//读取叠台的数据
rtRead(CLK:=ReadPointVelues , Q=> );
ftRead(CLK:=ReadPointVelues , Q=> );	
	IF rtRead.Q THEN
		mcReadMotionFunctionValues.Execute:=TRUE;
		CamTable3.pArray:=ADR(arrTableData);
		CamTable3.ArraySize:=SIZEOF(arrTableData);
		CamTable3.NoOfColumns:=2;
		CamTable3.NoOfRows:=3601;
		CamTable3.TableType:=10;	
	END_IF	
	 mcReadMotionFunctionValues1(
		  Execute:=                          mcReadMotionFunctionValues.Execute , 
		  CamTableID:=                   iTable , 
		  ValueSelectMask:=               1 ,
		  StartPosMaster:=               0 , 
		  EndPosMaster:=                360 , //360
		  Increment:=                       0.1 , 
		  Done=>                           arrReadPosDone , 
		  Busy=>mcReadMotionFunctionValues_Busy                              , 
		  Error=>mcReadMotionFunctionValues_Error                             , 
		  ErrorID=>mcReadMotionFunctionValues_ErrorID                         , 
		  CamTable:=                      CamTable3      );
	IF ftRead.Q THEN
		mcReadMotionFunctionValues.Execute:=FALSE;	
	END_IF	
//叠台中心点，主轴相位计算 fbCenterPoint
	Test_int:=REAL_TO_INT(fMainPos*10);
	FOR	i:=0 TO Test_int BY 1  DO
		IF (fbCenterPoint-0.15)< arrTableData[i,1] AND arrTableData[i,1]<(fbCenterPoint +0.15) THEN
			iFend:=i;
			Master_MidPos:=arrTableData[i,0];			
		END_IF		
	END_FOR
END_ACTION

ACTION Motion:
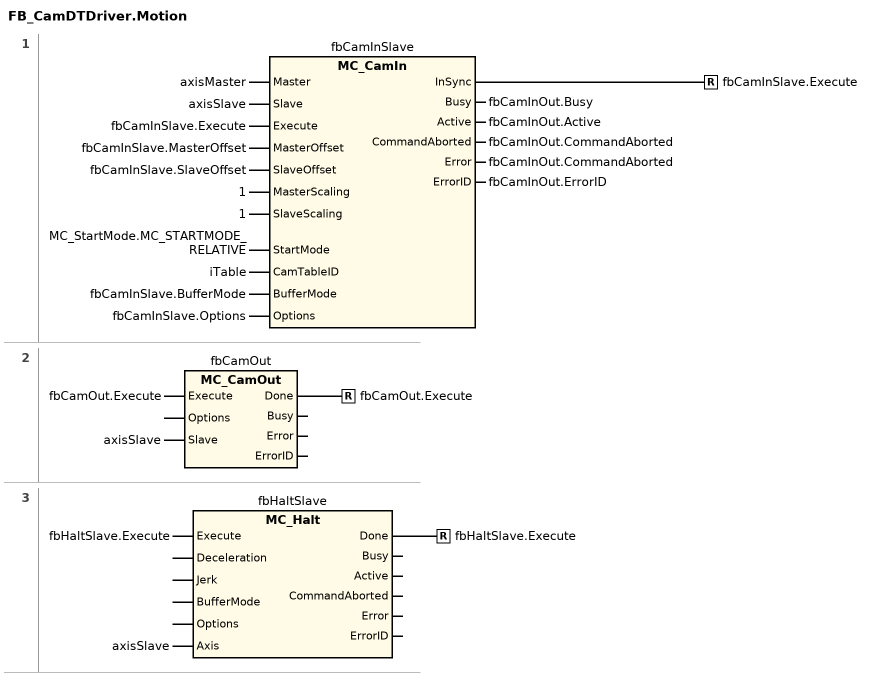
// NETWORK 1
fbCamInSlave(
    Master := axisMaster,
    Slave := axisSlave,
    Execute := fbCamInSlave.Execute,
    MasterOffset := fbCamInSlave.MasterOffset,
    SlaveOffset := fbCamInSlave.SlaveOffset,
    MasterScaling := 1,
    SlaveScaling := 1,
    StartMode := MC_StartMode.MC_STARTMODE_RELATIVE,
    CamTableID := iTable,
    BufferMode := fbCamInSlave.BufferMode,
    Options := fbCamInSlave.Options,
    Busy => fbCamInOut.Busy,
    Active => fbCamInOut.Active,
    CommandAborted => fbCamInOut.CommandAborted,
    Error => fbCamInOut.CommandAborted,
    ErrorID => fbCamInOut.ErrorID); // MC_CamIn
fbCamInSlave.Execute R= fbCamInSlave.InSync;

// NETWORK 2
fbCamOut(Execute := fbCamOut.Execute, Slave := axisSlave); // MC_CamOut
fbCamOut.Execute R= fbCamOut.Done;

// NETWORK 3
fbHaltSlave(Execute := fbHaltSlave.Execute, Axis := axisSlave); // MC_Halt
fbHaltSlave.Execute R= fbHaltSlave.Done;
END_ACTION

END_FUNCTION_BLOCK

// ---- P2POUs/BasicFunction/12_User2/FB_Rectify.TcPOU
FUNCTION_BLOCK FB_Rectify
VAR_INPUT
	
END_VAR
VAR_IN_OUT
     RecCtrl:     ST_RecCtrl;
END_VAR
VAR
   rtRec  :ARRAY[1..4] OF Tc2_Standard.R_TRIG;
END_VAR









rtRec[1](CLK:=RecCtrl.Cmd.bLock , Q=> );
rtRec[2](CLK:=RecCtrl.Cmd.bAuto , Q=> );
rtRec[3](CLK:=RecCtrl.Cmd.bManual , Q=> );
rtRec[4](CLK:=RecCtrl.Cmd.bCentre , Q=> );

IF rtRec[1].Q   THEN  //外部锁定
    RecCtrl.Io.boLock:=TRUE;
    RecCtrl.Io.boAuto:=FALSE;
    RecCtrl.Io.boManual:=FALSE;
    RecCtrl.Io.boCentre:=FALSE;
END_IF

IF rtRec[2].Q   THEN  //自动
    RecCtrl.Io.boLock:=FALSE;
    RecCtrl.Io.boAuto:=TRUE;
    RecCtrl.Io.boManual:=FALSE;
    RecCtrl.Io.boCentre:=FALSE;
END_IF

IF rtRec[3].Q   THEN  //手动
    RecCtrl.Io.boLock:=FALSE;
    RecCtrl.Io.boAuto:=FALSE;
    RecCtrl.Io.boManual:=TRUE;
    RecCtrl.Io.boCentre:=FALSE;
END_IF

IF rtRec[4].Q   THEN  //居中
    RecCtrl.Io.boLock:=FALSE;
    RecCtrl.Io.boAuto:=FALSE;
    RecCtrl.Io.boManual:=FALSE;
    RecCtrl.Io.boCentre:=TRUE;
END_IF


RecCtrl.Status.bError:=RecCtrl.Io.biError;
RecCtrl.Status.bRuning:=RecCtrl.Io.biCentre;

END_FUNCTION_BLOCK

// ---- P2POUs/BasicFunction/12_User2/Program_1.TcPOU
PROGRAM Program_1
VAR
Step0:INT;
TON1:Tc2_Standard.TON;
DemarcateStart,DemarcateDone,Demarcateing,CCDStart:BOOL;
	i: UINT;	
END_VAR

// scRecipe(iRecipe2:=iRecipe );
 
 TON1(IN:= , PT:=T#5S , Q=> , ET=> );//拍照延时复位


CASE Step0 OF
		0://等待CCD标定启动信号
		        P2M1_CCD.AnRec.Start.iPhotoDo:=0;
		        P2M1_CCD.AnRec.iDemarcatResult:=0;
			IF DemarcateStart THEN
				i:=0;//标定点位记数
			    P2M1_CCD.AnRec.Start.iPhotoDo:=1;
				DemarcateStart:=FALSE;//复位标定启动
				DemarcateDone:=FALSE;//CCD标定完成
				Demarcateing:=TRUE;//CCD标定中
				Step0:=5;
			END_IF
	5:
IF 		P2M1_CCD.AnRec.iDemarcatResult=1 AND  P2M1_CCD.AnRec.Start.iPhotoDo=0 THEN 
         P2M1_CCD.AnRec.iDemarcatResult:=0;
		 	i:=1;
			Step0:=10;
ELSIF 	P2M1_CCD.AnRec.iDemarcatResult=2 AND  P2M1_CCD.AnRec.Start.iPhotoDo=0 THEN 
	P2M1_CCD.AnRec.iDemarcatResult:=0;
	Step0:=999;
END_IF
		10://判断CCD标定走到第几个点位
					IF  i=1 THEN
									arrAxisPar[P2M1_Axise.AxisName.AndeviationX1].arrTargetPoint[3]:=arrAxisPar[P2M1_Axise.AxisName.AndeviationX1].arrTargetPoint[1];//+(103.94*COS(DEG_TO_RAD(CCD_W+225))-103.94*COS(DEG_TO_RAD(225))); 
									arrAxisPar[P2M1_Axise.AxisName.AndeviationX2].arrTargetPoint[3]:=arrAxisPar[P2M1_Axise.AxisName.AndeviationX2].arrTargetPoint[1];//+(103.94*SIN(DEG_TO_RAD(CCD_W+315))-103.94*COS(DEG_TO_RAD(315)));
									arrAxisPar[P2M1_Axise.AxisName.AndeviationY].arrTargetPoint[3]:=arrAxisPar[P2M1_Axise.AxisName.AndeviationY].arrTargetPoint[1];//+(103.94*COS(DEG_TO_RAD(CCD_W+135))-103.94*COS(DEG_TO_RAD(135)));	
									//i:=i+1;
									Step0:=20;
					ELSIF i=2 THEN
									arrAxisPar[P2M1_Axise.AxisName.AndeviationX1].arrTargetPoint[3]:=arrAxisPar[P2M1_Axise.AxisName.AndeviationX1].arrTargetPoint[1]+4;//+(103.94*COS(DEG_TO_RAD(CCD_W+225))-103.94*COS(DEG_TO_RAD(225))); 
									arrAxisPar[P2M1_Axise.AxisName.AndeviationX2].arrTargetPoint[3]:=arrAxisPar[P2M1_Axise.AxisName.AndeviationX2].arrTargetPoint[1]+4;//+(103.94*SIN(DEG_TO_RAD(CCD_W+315))-103.94*COS(DEG_TO_RAD(315)));
									arrAxisPar[P2M1_Axise.AxisName.AndeviationY].arrTargetPoint[3]:=arrAxisPar[P2M1_Axise.AxisName.AndeviationY].arrTargetPoint[1];//+(103.94*COS(DEG_TO_RAD(CCD_W+135))-103.94*COS(DEG_TO_RAD(135)));
									//i:=i+1;
									Step0:=20;
					ELSIF i=3 THEN
									arrAxisPar[P2M1_Axise.AxisName.AndeviationX1].arrTargetPoint[3]:=arrAxisPar[P2M1_Axise.AxisName.AndeviationX1].arrTargetPoint[1]+4;//+(103.94*COS(DEG_TO_RAD(CCD_W+225))-103.94*COS(DEG_TO_RAD(225))); 
									arrAxisPar[P2M1_Axise.AxisName.AndeviationX2].arrTargetPoint[3]:=arrAxisPar[P2M1_Axise.AxisName.AndeviationX2].arrTargetPoint[1]+4;//+(103.94*SIN(DEG_TO_RAD(CCD_W+315))-103.94*COS(DEG_TO_RAD(315)));
									arrAxisPar[P2M1_Axise.AxisName.AndeviationY].arrTargetPoint[3]:=arrAxisPar[P2M1_Axise.AxisName.AndeviationY].arrTargetPoint[1]+4;//+(103.94*COS(DEG_TO_RAD(CCD_W+135))-103.94*COS(DEG_TO_RAD(135)));	
									//i:=i+1;
									Step0:=20;									
					ELSIF i=4 THEN
								arrAxisPar[P2M1_Axise.AxisName.AndeviationX1].arrTargetPoint[3]:=arrAxisPar[P2M1_Axise.AxisName.AndeviationX1].arrTargetPoint[1];//+(103.94*COS(DEG_TO_RAD(CCD_W+225))-103.94*COS(DEG_TO_RAD(225))); 
								arrAxisPar[P2M1_Axise.AxisName.AndeviationX2].arrTargetPoint[3]:=arrAxisPar[P2M1_Axise.AxisName.AndeviationX2].arrTargetPoint[1];//+(103.94*SIN(DEG_TO_RAD(CCD_W+315))-103.94*COS(DEG_TO_RAD(315)));
								arrAxisPar[P2M1_Axise.AxisName.AndeviationY].arrTargetPoint[3]:=arrAxisPar[P2M1_Axise.AxisName.AndeviationY].arrTargetPoint[1]+4;//+(103.94*COS(DEG_TO_RAD(CCD_W+135))-103.94*COS(DEG_TO_RAD(135)));	
								//i:=i+1;
								Step0:=20;		
					ELSIF i=5 THEN
								arrAxisPar[P2M1_Axise.AxisName.AndeviationX1].arrTargetPoint[3]:=arrAxisPar[P2M1_Axise.AxisName.AndeviationX1].arrTargetPoint[1]-4;//+(103.94*COS(DEG_TO_RAD(CCD_W+225))-103.94*COS(DEG_TO_RAD(225))); 
								arrAxisPar[P2M1_Axise.AxisName.AndeviationX2].arrTargetPoint[3]:=arrAxisPar[P2M1_Axise.AxisName.AndeviationX2].arrTargetPoint[1]-4;//+(103.94*SIN(DEG_TO_RAD(CCD_W+315))-103.94*COS(DEG_TO_RAD(315)));
								arrAxisPar[P2M1_Axise.AxisName.AndeviationY].arrTargetPoint[3]:=arrAxisPar[P2M1_Axise.AxisName.AndeviationY].arrTargetPoint[1]+4;//+(103.94*COS(DEG_TO_RAD(CCD_W+135))-103.94*COS(DEG_TO_RAD(135)));	
							//	i:=i+1;
								Step0:=20;		
					ELSIF i=6 THEN
								arrAxisPar[P2M1_Axise.AxisName.AndeviationX1].arrTargetPoint[3]:=arrAxisPar[P2M1_Axise.AxisName.AndeviationX1].arrTargetPoint[1]-4;//+(103.94*COS(DEG_TO_RAD(CCD_W+225))-103.94*COS(DEG_TO_RAD(225))); 
								arrAxisPar[P2M1_Axise.AxisName.AndeviationX2].arrTargetPoint[3]:=arrAxisPar[P2M1_Axise.AxisName.AndeviationX2].arrTargetPoint[1]-4;//+(103.94*SIN(DEG_TO_RAD(CCD_W+315))-103.94*COS(DEG_TO_RAD(315)));
								arrAxisPar[P2M1_Axise.AxisName.AndeviationY].arrTargetPoint[3]:=arrAxisPar[P2M1_Axise.AxisName.AndeviationY].arrTargetPoint[1];//+(103.94*COS(DEG_TO_RAD(CCD_W+135))-103.94*COS(DEG_TO_RAD(135)));	
								//i:=i+1;
								Step0:=20;		
					ELSIF i=7 THEN
									arrAxisPar[P2M1_Axise.AxisName.AndeviationX1].arrTargetPoint[3]:=arrAxisPar[P2M1_Axise.AxisName.AndeviationX1].arrTargetPoint[1]-4;//+(103.94*COS(DEG_TO_RAD(CCD_W+225))-103.94*COS(DEG_TO_RAD(225))); 
									arrAxisPar[P2M1_Axise.AxisName.AndeviationX2].arrTargetPoint[3]:=arrAxisPar[P2M1_Axise.AxisName.AndeviationX2].arrTargetPoint[1]-4;//+(103.94*SIN(DEG_TO_RAD(CCD_W+315))-103.94*COS(DEG_TO_RAD(315)));
									arrAxisPar[P2M1_Axise.AxisName.AndeviationY].arrTargetPoint[3]:=arrAxisPar[P2M1_Axise.AxisName.AndeviationY].arrTargetPoint[1]-4;//+(103.94*COS(DEG_TO_RAD(CCD_W+135))-103.94*COS(DEG_TO_RAD(135)));
								//	i:=i+1;
									Step0:=20;		
					ELSIF i=8 THEN
									arrAxisPar[P2M1_Axise.AxisName.AndeviationX1].arrTargetPoint[3]:=arrAxisPar[P2M1_Axise.AxisName.AndeviationX1].arrTargetPoint[1];//+(103.94*COS(DEG_TO_RAD(CCD_W+225))-103.94*COS(DEG_TO_RAD(225))); 
									arrAxisPar[P2M1_Axise.AxisName.AndeviationX2].arrTargetPoint[3]:=arrAxisPar[P2M1_Axise.AxisName.AndeviationX2].arrTargetPoint[1];//+(103.94*SIN(DEG_TO_RAD(CCD_W+315))-103.94*COS(DEG_TO_RAD(315)));
									arrAxisPar[P2M1_Axise.AxisName.AndeviationY].arrTargetPoint[3]:=arrAxisPar[P2M1_Axise.AxisName.AndeviationY].arrTargetPoint[1]-4;//+(103.94*COS(DEG_TO_RAD(CCD_W+135))-103.94*COS(DEG_TO_RAD(135)));	
									//i:=i+1;
									Step0:=20;		
					ELSIF i=9 THEN
								arrAxisPar[P2M1_Axise.AxisName.AndeviationX1].arrTargetPoint[3]:=arrAxisPar[P2M1_Axise.AxisName.AndeviationX1].arrTargetPoint[1]+4;//+(103.94*COS(DEG_TO_RAD(CCD_W+225))-103.94*COS(DEG_TO_RAD(225))); 
								arrAxisPar[P2M1_Axise.AxisName.AndeviationX2].arrTargetPoint[3]:=arrAxisPar[P2M1_Axise.AxisName.AndeviationX2].arrTargetPoint[1]+4;//+(103.94*SIN(DEG_TO_RAD(CCD_W+315))-103.94*COS(DEG_TO_RAD(315)));
								arrAxisPar[P2M1_Axise.AxisName.AndeviationY].arrTargetPoint[3]:=arrAxisPar[P2M1_Axise.AxisName.AndeviationY].arrTargetPoint[1]-4;//+(103.94*COS(DEG_TO_RAD(CCD_W+135))-103.94*COS(DEG_TO_RAD(135)));	
								//i:=i+1;
								Step0:=20;		
					ELSIF i=10 THEN
								arrAxisPar[P2M1_Axise.AxisName.AndeviationX1].arrTargetPoint[3]:=arrAxisPar[P2M1_Axise.AxisName.AndeviationX1].arrTargetPoint[1];//+(103.94*COS(DEG_TO_RAD(CCD_W+225))-103.94*COS(DEG_TO_RAD(225))); 
								arrAxisPar[P2M1_Axise.AxisName.AndeviationX2].arrTargetPoint[3]:=arrAxisPar[P2M1_Axise.AxisName.AndeviationX2].arrTargetPoint[1];//+(103.94*SIN(DEG_TO_RAD(CCD_W+315))-103.94*COS(DEG_TO_RAD(315)));
								arrAxisPar[P2M1_Axise.AxisName.AndeviationY].arrTargetPoint[3]:=arrAxisPar[P2M1_Axise.AxisName.AndeviationY].arrTargetPoint[1];//+(103.94*COS(DEG_TO_RAD(CCD_W+135))-103.94*COS(DEG_TO_RAD(135)));	
								//i:=i+1;
								Step0:=20;		
					ELSIF i=11 THEN
								arrAxisPar[P2M1_Axise.AxisName.AndeviationX1].arrTargetPoint[3]:=arrAxisPar[P2M1_Axise.AxisName.AndeviationX1].arrTargetPoint[1]+(103.94*COS(DEG_TO_RAD(2+225))-103.94*COS(DEG_TO_RAD(225))); 
								arrAxisPar[P2M1_Axise.AxisName.AndeviationX2].arrTargetPoint[3]:=arrAxisPar[P2M1_Axise.AxisName.AndeviationX2].arrTargetPoint[1]+(103.94*SIN(DEG_TO_RAD(2+315))-103.94*COS(DEG_TO_RAD(315)));
								arrAxisPar[P2M1_Axise.AxisName.AndeviationY].arrTargetPoint[3]:=arrAxisPar[P2M1_Axise.AxisName.AndeviationY].arrTargetPoint[1]+(103.94*COS(DEG_TO_RAD(2+135))-103.94*COS(DEG_TO_RAD(135)));	
								//i:=i+1;
								Step0:=20;		
					ELSIF i=12 THEN
									arrAxisPar[P2M1_Axise.AxisName.AndeviationX1].arrTargetPoint[3]:=arrAxisPar[P2M1_Axise.AxisName.AndeviationX1].arrTargetPoint[1]+(103.94*COS(DEG_TO_RAD(1+225))-103.94*COS(DEG_TO_RAD(225))); 
									arrAxisPar[P2M1_Axise.AxisName.AndeviationX2].arrTargetPoint[3]:=arrAxisPar[P2M1_Axise.AxisName.AndeviationX2].arrTargetPoint[1]+(103.94*SIN(DEG_TO_RAD(1+315))-103.94*COS(DEG_TO_RAD(315)));
									arrAxisPar[P2M1_Axise.AxisName.AndeviationY].arrTargetPoint[3]:=arrAxisPar[P2M1_Axise.AxisName.AndeviationY].arrTargetPoint[1]+(103.94*COS(DEG_TO_RAD(1+135))-103.94*COS(DEG_TO_RAD(135)));
									//i:=i+1;
									Step0:=20;		
					
					ELSIF i=130 THEN
									arrAxisPar[P2M1_Axise.AxisName.AndeviationX1].arrTargetPoint[3]:=arrAxisPar[P2M1_Axise.AxisName.AndeviationX1].arrTargetPoint[1];//+(103.94*COS(DEG_TO_RAD(CCD_W+225))-103.94*COS(DEG_TO_RAD(225))); 
									arrAxisPar[P2M1_Axise.AxisName.AndeviationX2].arrTargetPoint[3]:=arrAxisPar[P2M1_Axise.AxisName.AndeviationX2].arrTargetPoint[1];//+(103.94*SIN(DEG_TO_RAD(CCD_W+315))-103.94*COS(DEG_TO_RAD(315)));
									arrAxisPar[P2M1_Axise.AxisName.AndeviationY].arrTargetPoint[3]:=arrAxisPar[P2M1_Axise.AxisName.AndeviationY].arrTargetPoint[1];//+(103.94*COS(DEG_TO_RAD(CCD_W+135))-103.94*COS(DEG_TO_RAD(135)));	
									//i:=i+1;
									Step0:=20;		
					ELSIF i=140 THEN
								arrAxisPar[P2M1_Axise.AxisName.AndeviationX1].arrTargetPoint[3]:=arrAxisPar[P2M1_Axise.AxisName.AndeviationX1].arrTargetPoint[1]+(103.94*COS(DEG_TO_RAD(-1+225))-103.94*COS(DEG_TO_RAD(225))); 
								arrAxisPar[P2M1_Axise.AxisName.AndeviationX2].arrTargetPoint[3]:=arrAxisPar[P2M1_Axise.AxisName.AndeviationX2].arrTargetPoint[1]+(103.94*SIN(DEG_TO_RAD(-1+315))-103.94*COS(DEG_TO_RAD(315)));
								arrAxisPar[P2M1_Axise.AxisName.AndeviationY].arrTargetPoint[3]:=arrAxisPar[P2M1_Axise.AxisName.AndeviationY].arrTargetPoint[1]+(103.94*COS(DEG_TO_RAD(-1+135))-103.94*COS(DEG_TO_RAD(135)));	
								//i:=i+1;
								Step0:=20;		
					ELSIF i=150 THEN
								arrAxisPar[P2M1_Axise.AxisName.AndeviationX1].arrTargetPoint[3]:=arrAxisPar[P2M1_Axise.AxisName.AndeviationX1].arrTargetPoint[1]+(103.94*COS(DEG_TO_RAD(-2+225))-103.94*COS(DEG_TO_RAD(225))); 
								arrAxisPar[P2M1_Axise.AxisName.AndeviationX2].arrTargetPoint[3]:=arrAxisPar[P2M1_Axise.AxisName.AndeviationX2].arrTargetPoint[1]+(103.94*SIN(DEG_TO_RAD(-2+315))-103.94*COS(DEG_TO_RAD(315)));
								arrAxisPar[P2M1_Axise.AxisName.AndeviationY].arrTargetPoint[3]:=arrAxisPar[P2M1_Axise.AxisName.AndeviationY].arrTargetPoint[1]+(103.94*COS(DEG_TO_RAD(-2+135))-103.94*COS(DEG_TO_RAD(135)));	
								//i:=i+1;
								Step0:=20;		
					ELSIF i=160 THEN
								arrAxisPar[P2M1_Axise.AxisName.AndeviationX1].arrTargetPoint[3]:=arrAxisPar[P2M1_Axise.AxisName.AndeviationX1].arrTargetPoint[1];//+(103.94*COS(DEG_TO_RAD(CCD_W+225))-103.94*COS(DEG_TO_RAD(225))); 
								arrAxisPar[P2M1_Axise.AxisName.AndeviationX2].arrTargetPoint[3]:=arrAxisPar[P2M1_Axise.AxisName.AndeviationX2].arrTargetPoint[1];//+(103.94*SIN(DEG_TO_RAD(CCD_W+315))-103.94*COS(DEG_TO_RAD(315)));
								arrAxisPar[P2M1_Axise.AxisName.AndeviationY].arrTargetPoint[3]:=arrAxisPar[P2M1_Axise.AxisName.AndeviationY].arrTargetPoint[1];//+(103.94*COS(DEG_TO_RAD(CCD_W+135))-103.94*COS(DEG_TO_RAD(135)));		
								//i:=i+1;
								Step0:=20;													
					END_IF	
		(*
	FOR i:=0 TO 15 DO 
					arrAxisPar[P2M1_Axise.AxisName.AndeviationX1].arrTargetPoint[3]:=arrAxisPar[P2M1_Axise.AxisName.AndeviationX1].arrTargetPoint[1]+(103.94*COS(DEG_TO_RAD(CCD_W+225))-103.94*COS(DEG_TO_RAD(225))); 
					arrAxisPar[P2M1_Axise.AxisName.AndeviationX2].arrTargetPoint[3]:=arrAxisPar[P2M1_Axise.AxisName.AndeviationX2].arrTargetPoint[1]+(103.94*SIN(DEG_TO_RAD(CCD_W+315))-103.94*COS(DEG_TO_RAD(315)));
					arrAxisPar[P2M1_Axise.AxisName.AndeviationY].arrTargetPoint[3]:=arrAxisPar[P2M1_Axise.AxisName.AndeviationY].arrTargetPoint[1]+(103.94*COS(DEG_TO_RAD(CCD_W+135))-103.94*COS(DEG_TO_RAD(135)));				
	END_FOR
	*)
	20:

	P2M1_CCD.AnRec.Start.iPhotoDo:=1; 
	Step0:=25;				
	25:
IF P2M1_CCD.AnRec.Start.iPhotoDo=0  AND P2M1_CCD.AnRec.iDemarcatResult=1     THEN
	P2M1_CCD.AnRec.iDemarcatResult:=0; 
	Step0:=30;		
ELSIF P2M1_CCD.AnRec.Start.iPhotoDo=0  AND P2M1_CCD.AnRec.iDemarcatResult=2     THEN	
	P2M1_CCD.AnRec.iDemarcatResult:=0;
	Step0:=999;		
 END_IF
	30://移动至标定位
			IF arrAxisCtrl[P2M1_Axise.AxisName.AndeviationX1].Status.Homed OR (arrAxisCtrl[P2M1_Axise.AxisName.AndeviationX1].Status.NoMoving AND NOT arrAxisCtrl[P2M1_Axise.AxisName.AndeviationX1].Status.Error )THEN
						IF arrAxisCtrl[P2M1_Axise.AxisName.AndeviationX1].Cmd.arrbRealPoint[3] THEN
							;//arrAxisCtrl[P2M1_Axise.AxisName.AndeviationX1].Cmd.iGoSetPos:=0;
						ELSE
							arrAxisCtrl[P2M1_Axise.AxisName.AndeviationX1].Cmd.iGoSetPos:=3;
						END_IF 
			END_IF
			IF arrAxisCtrl[P2M1_Axise.AxisName.AndeviationX2].Status.Homed OR  (arrAxisCtrl[P2M1_Axise.AxisName.AndeviationX2].Status.NoMoving AND NOT arrAxisCtrl[P2M1_Axise.AxisName.AndeviationX2].Status.Error) THEN
						IF arrAxisCtrl[P2M1_Axise.AxisName.AndeviationX2].Cmd.arrbRealPoint[3] THEN
						;	//arrAxisCtrl[P2M1_Axise.AxisName.AndeviationX2].Cmd.iGoSetPos:=0;
						ELSE
							arrAxisCtrl[P2M1_Axise.AxisName.AndeviationX2].Cmd.iGoSetPos:=3;
						END_IF
			END_IF	
			IF arrAxisCtrl[P2M1_Axise.AxisName.AndeviationY].Status.Homed OR (arrAxisCtrl[P2M1_Axise.AxisName.AndeviationY].Status.NoMoving AND NOT arrAxisCtrl[P2M1_Axise.AxisName.AndeviationY].Status.Error) THEN
						IF arrAxisCtrl[P2M1_Axise.AxisName.AndeviationY].Cmd.arrbRealPoint[3] THEN
							;//arrAxisCtrl[P2M1_Axise.AxisName.AndeviationY].Cmd.iGoSetPos:=0;
						ELSE
							arrAxisCtrl[P2M1_Axise.AxisName.AndeviationY].Cmd.iGoSetPos:=3;
						END_IF
			END_IF
			IF  arrAxisCtrl[P2M1_Axise.AxisName.AndeviationX1].Cmd.arrbRealPoint[3]  AND 	arrAxisCtrl[P2M1_Axise.AxisName.AndeviationY].Cmd.arrbRealPoint[3] AND  arrAxisCtrl[P2M1_Axise.AxisName.AndeviationY].Cmd.arrbRealPoint[3] THEN
				TON1.IN:=TRUE;	
            Step0:=40;
			END_IF		
	40://延时拍照
			IF 	 TON1.Q  THEN
				TON1.IN:=FALSE;	
				i:=i+1;
				Step0:=50;
				END_IF
 
			
	50://
			IF i>=13 THEN	
				Step0:=60;
			ELSE
				Step0:=10;
			END_IF	
	60:
	P2M1_CCD.AnRec.Start.iPhotoDo:=1; 
	Step0:=70;		
70:
IF P2M1_CCD.AnRec.Start.iPhotoDo=0  AND P2M1_CCD.AnRec.iDemarcatResult=1     THEN
	P2M1_CCD.AnRec.iDemarcatResult:=0; 
	DemarcateDone:=TRUE;//CCD标定完成
	Demarcateing:=FALSE;//CCD标定中
	Step0:=666;		
ELSIF P2M1_CCD.AnRec.Start.iPhotoDo=0  AND P2M1_CCD.AnRec.iDemarcatResult=2     THEN	
	P2M1_CCD.AnRec.iDemarcatResult:=0;
	Step0:=999;		
 END_IF				
END_CASE

END_PROGRAM

// ---- P2POUs/POUS/FunctionTest.TcPOU
PROGRAM FunctionTest
VAR





 fbCamPTPTest   :FB_CamPTPTest;

 fbCamPTPTest2   :FB_CamPTPTestV2;
	bMoveExecute: BOOL;

    fbCamTrapezoid:FB_CamTrapezoid;

	bMoveExecute2: BOOL;
END_VAR

//P2M1_Auto();
//P2M2_Auto();
//P2M3_Auto();

TEST();

ACTION P2M1_Auto:
// 1号叠台自动
//P2M1_program(Sys_Control:=P2_sysControl , Mach_Control:=P2M1_MachCtrl , arrCyNo:=P2M1_CycNo , AxiseNo:=P2M1_Axise , TableNo:=P2M1_TableNo,Par:=P2M1_Par );
END_ACTION

ACTION P2M2_Auto:
// 2号叠台自动
//P2M2_program(Sys_Control:=P2_sysControl , Mach_Control:=P2M2_MachCtrl , arrCyNo:=P2M2_CycNo , AxiseNo:=P2M2_Axise ,TableNo:=P2M2_TableNo, Par:=P2M2_Par );
END_ACTION

ACTION P2M3_Auto:
// 3号叠台自动
//P2M3_program(Sys_Control:=P2_sysControl , Mach_Control:=P2M3_MachCtrl , arrCyNo:=P2M3_CycNo , AxiseNo:=P2M3_Axise ,TableNo:=P2M3_TableNo ,Par:=P2M3_Par );
END_ACTION

ACTION TEST:



fbCamPTPTest(
	bMoveCamAbsExecute:=fbCamPTPTest.bMoveCamAbsExecute , 
	Reset:=                          stSysState.bReset  ,  
	iTable:=                         29   , 
	fTagatPos:=                  360 , 
	fTagatTime:=                 fbCamPTPTest.fTagatTime , 
    axisTimer:=                  arrAxis[140]  , 
	axisSlave:=                   arrAxis[141]  , 
	
	bCreatTableDone=> , 
	bCreatTableError=> , 
	bError=> , 
	bReady=> , 
	Done=> , 
	bInSync=> );

fbCamPTPTest.bCreatTableDone;
fbCamPTPTest.bCreatTableError;
fbCamPTPTest.bError;
fbCamPTPTest.bReady;
fbCamPTPTest.Done;
fbCamPTPTest.bInSync;




fbCamPTPTest2(
	fTagatPos:=                 360, 
	fTagatTime:=               fbCamPTPTest2.fTagatTime        , 
	fConVelPercentage:=    fbCamPTPTest2.fConVelPercentage      , 
	bMoveExecute:=          bMoveExecute , 
	axisSlave:=                   arrAxis[141] , 
	Done=> , 
	Busy=> , 
	Alm=> );
fbCamPTPTest2.Done;
fbCamPTPTest2.Busy;
fbCamPTPTest2.Alm;



fbCamTrapezoid(
	fTagatPos:=             360 , 
	fTagatTime:=           fbCamTrapezoid.fTagatTime  , 
	fConVelPercentage:=fbCamTrapezoid.fConVelPercentage , 
	bMoveExecute:=      bMoveExecute2 , 
	axisSlave:=            arrAxis[141] , 
	Done=> , 
	Busy=> , 
	Alm=> );

fbCamTrapezoid.Done;
fbCamTrapezoid.Busy;
fbCamTrapezoid.Alm;
END_ACTION

END_PROGRAM

// ---- P3POUs/P3FB/CS_SetpMoterV2.TcPOU
FUNCTION_BLOCK CS_SetpMoterV2
VAR_INPUT
END_VAR
VAR_OUTPUT
END_VAR
VAR
	
	
END_VAR

VAR_IN_OUT
stSetpMotor:ST_SetpMotor;//电芯出料步进电机	
END_VAR
	

VAR
iSensorCount: INT;
//R_TRIG10:R_TRIG;
//F_TRIG10:F_TRIG;
R_trig20:R_TRIG;
R_trig21:R_TRIG;
R_trig23:R_TRIG;
R_trig22:R_TRIG;
TON50:TON;
TON51:TON;
TON52:TON;
TON53:TON;
//TON54:TON;
iSetp3:INT;   //电芯转移流程


END_VAR

(*********************步进电机控制*****************************)
//步进点动
stSetpMotor.bo_Up:= ( stSetpMotor.bJog_Up AND NOT stSetpMotor.biUpSensor) OR  ( stSetpMotor.bJog_Down AND NOT stSetpMotor.biDownSensor ); //步进启动   
stSetpMotor.bo_Down:=stSetpMotor.bJog_Down AND NOT stSetpMotor.biDownSensor ;   //步进方向选择，默认0为上升   

//步进回原点
iSensorCount:=BOOL_TO_INT(stSetpMotor.biUpSensor)+ BOOL_TO_INT(stSetpMotor.biRefSensor)+ BOOL_TO_INT(stSetpMotor.biDownSensor);
R_trig20(CLK:=stSetpMotor.bHome , Q=> );
IF R_trig20.Q  AND iSensorCount<=1 THEN
   iSetp3:=88;
   stSetpMotor.bHome:=FALSE;
   stSetpMotor.HomeDone:=FALSE;
END_IF

R_trig21(CLK:=stSetpMotor.bGoWorkPos , Q=> ); //GO工作位置  
IF R_trig21.Q  THEN  //AND iSensorCount<=1
   stSetpMotor.bJog_Down:=FALSE;
   stSetpMotor.bJog_Up:=FALSE;
   iSetp3:=99;	
   //stSetpMotor.HomeDone:=FALSE;
   stSetpMotor.bGoWorkPos:=FALSE;
   stSetpMotor.WorkPosDone:=FALSE;
END_IF

R_trig23(CLK:=stSetpMotor.bLeaveWorkPos , Q=> ); //离开工作位置  
IF R_trig23.Q  THEN  //AND iSensorCount<=1
   stSetpMotor.bJog_Down:=FALSE;
     stSetpMotor.bJog_Up:=FALSE;
    iSetp3:=97;	
	//stSetpMotor.HomeDone:=FALSE;
   stSetpMotor.bLeaveWorkPos:=FALSE;
   stSetpMotor.WorkPosDone:=FALSE;
END_IF

TON50(IN:= , PT:=T#20MS , Q=> , ET=> );  //感应原点后延时
TON51(IN:= , PT:=T#20MS , Q=> , ET=> );  //对射感应原点后延时
TON52(IN:= , PT:=T#10S , Q=> , ET=> );  //感应电芯报警
TON53(IN:= , PT:=T#300MS , Q=> , ET=> );  //感
R_trig22(CLK:=iSensorCount=1 , Q=> );  


CASE iSetp3 OF   	
88:  
   IF stSetpMotor.biSensor  AND stSetpMotor.bJog_Up THEN  //本来就在原点  回原完成
	   TON50.IN:=TRUE; 
	   TON52.IN:=FALSE;
	   IF TON50.Q THEN
		   stSetpMotor.HomeDone:=TRUE;
		   stSetpMotor.bJog_Down:=FALSE;
		   stSetpMotor.bJog_Up:=FALSE; 		   
		   TON50.IN:=FALSE;  
		   iSetp3:=666;   
	   END_IF
   ELSIF  stSetpMotor.biDownSensor THEN  
	     iSetp3:=100; 
   ELSIF  stSetpMotor.biUpSensor THEN 	   
	      iSetp3:=200;    
   ELSE                //没在任何感应 
       iSetp3:=200;    //默认往参考点回原点
   END_IF
   
100:  //上升
	   stSetpMotor.bJog_Down:=FALSE;
	   stSetpMotor.bJog_Up:=TRUE;      //下限位 往上  碰到 mid2停
	    IF stSetpMotor.biSensor THEN
		  iSetp3:=88;	
		END_IF   
200:   //下降
	   stSetpMotor.bJog_Down:=TRUE;
	   stSetpMotor.bJog_Up:=FALSE; 
	   IF  R_trig22.Q THEN   //下将过程中碰到限位
		   iSetp3:=88;	
			//stSetpMotor.HomeDone:=TRUE; 
	   END_IF   
  
(*************************对射位置***********************)   
99:    //在原位先上升    
	   stSetpMotor.bJog_Down:=FALSE;
	    stSetpMotor.bJog_Up:=TRUE;  
		TON52.IN:=TRUE;
		 iSetp3:=300;    	   
300: //对射检测
	 IF stSetpMotor.biUpSensor  THEN 
	    stSetpMotor.bJog_Down:=TRUE;
	    stSetpMotor.bJog_Up:=FALSE; 
	 END_IF

		IF stSetpMotor.biSensor   THEN //stSetpMotor.biSensor
		   TON51.IN:=TRUE; 
		   IF TON51.Q THEN 
			   stSetpMotor.WorkPosDone:=TRUE;
               stSetpMotor.bJog_Down:=FALSE;
			   stSetpMotor.bJog_Up:=FALSE; 
		       TON51.IN:=FALSE; 
			   iSetp3:=666;   
			END_IF   	
		END_IF
		
(**************************离开对射位置********************************)  		
97:     
     IF  NOT stSetpMotor.bJog_Down AND NOT stSetpMotor.bJog_Up   THEN //升降轴上升到位 
		 stSetpMotor.bJog_Down:=TRUE;
		 stSetpMotor.bJog_Up:=FALSE;
         TON53.IN:=TRUE;
		 iSetp3:=400; 
	 END_IF		
		
400:  //步进电机回原位
	     IF TON53.Q AND NOT stSetpMotor.biSensor THEN//stSetpMotor.biSensor
		   stSetpMotor.WorkPosDone:=TRUE;
		    stSetpMotor.bJog_Down:=FALSE;
		    stSetpMotor.bJog_Up:=FALSE;	 
		     TON53.IN:=FALSE;
		   iSetp3:=666; 
		 END_IF
	     IF  stSetpMotor.biRefSensor OR stSetpMotor.biDownSensor  THEN
		     stSetpMotor.bJog_Down:=FALSE;
		      stSetpMotor.bJog_Up:=FALSE;	
             TON53.IN:=FALSE; 
		   // bAlarm:=TRUE;  
            stSetpMotor.bPoleFull:=TRUE;  
		    iSetp3:=666; 
		 END_IF							
END_CASE

END_FUNCTION_BLOCK

// ---- P3POUs/P3FB/FB_CSP_Velo_Torque.TcPOU
FUNCTION_BLOCK FB_CSP_Velo_Torque

VAR_IN_OUT
	Start_Torque			:BOOL	;//控制命令
	Axis : Axis_Ref;
	
END_VAR

VAR_INPUT
	
	Reset					:BOOL	;//复位
	Target_Torque			:REAL	;//设定压力
	Actual_Torque			:REAL	;//实际压力-从压力传感器获取
	DeadZone				:REAL	;//死区范围
	Hold_Time				:TIME	;//保压时间
	InitPosition			:REAL	;//初始位置
	StartPressPosition		:REAL	;//预压起始位置
	MaxPressPosition		:REAL	;//最大下压位置
	Press_Fast_xs:REAL;    //快速系数
	Press_Slow_xs:REAL;   //慢速系数
	Press_condition :BOOL;
	Option : ST_TorqueMotion ;	
END_VAR

VAR_OUTPUT
	Done				: BOOL		;//完成
	Busy				: BOOL		;//执行中
	Pressing			: BOOL		;//压合中
	CurrentPressTime 	: TIME;		;//实时压合时间
	HoldOK				: BOOL		;//保压中
	Error				: BOOL		;//热压超时报警
	ErrorID				: UDINT		;//报警ID
	ErrorMessage		: STRING	;//报警消息
	Error1				: BOOL		;//安全条件不满足不在报警
	BlowPermit			:BOOL;//吹气允许
END_VAR


VAR 	
	eWorkStep: INT;
	rtStart: R_trig;
	
	MoveAbs : MC_MoveAbsolute ;
	MoveVel : MC_MoveVelocity ;
	mcStop : MC_Halt;
	fPIDVelocity: LREAL;
	eTorqueStep: INT;
	bStart: BOOL;
	DeadZone_Min: REAL;
	DeadZone_Max: REAL;
	tonHoldPress: Ton;
	ErrorTorque: REAL;
	EnablePID: BOOL;
	eErrorStep: INT;
	error_ton :Tc2_Standard.TON;
	Stop_ton :Tc2_Standard.TON;
    Axis1_TON :Tc2_Standard.TON;
	tOutTime:TON;//超时
END_VAR

Act01_Status();

//死区范围
DeadZone_Min := Target_Torque - DeadZone ;
DeadZone_Max := Target_Torque + DeadZone ;

//保压计时
tonHoldPress(IN:= , PT:=Hold_Time, Q=> , ET=> );

IF  Error AND Reset AND eWorkStep<>0  AND ABS(Axis.NcToPlc.ActPos-InitPosition)<0.01THEN
	eWorkStep := 0;
	eTorqueStep := 0;
	EnablePID := FALSE;
	MoveVel.Execute := FALSE;
	tonHoldPress.IN := FALSE;
	HoldOK := FALSE;
	Busy := FALSE;
	Pressing := FALSE;
ELSE
	ErrorMessage := '';
	ErrorID := 0;
	


END_IF

IF Reset THEN
	Error  := FALSE;
	Error1 := FALSE;
	ErrorMessage := '';
	ErrorID := 0;
END_IF

Act02_ToqueMove();
Act10_Auto();
Act00_CallFB();

ACTION Act00_CallFB:
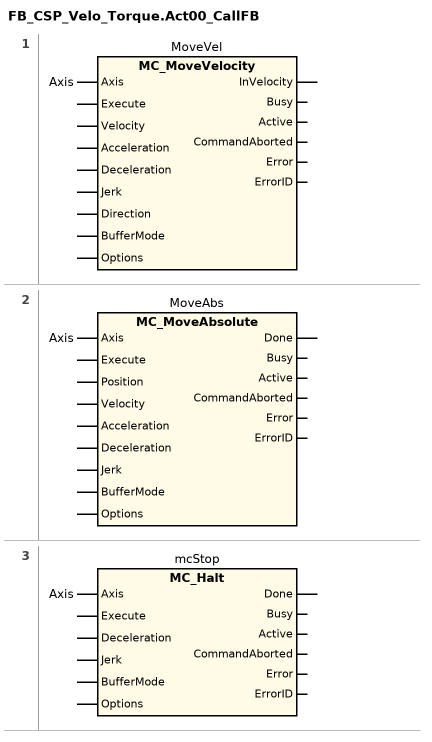
// NETWORK 1
MoveVel(Axis := Axis); // MC_MoveVelocity

// NETWORK 2
MoveAbs(Axis := Axis); // MC_MoveAbsolute

// NETWORK 3
mcStop(Axis := Axis); // MC_Halt
END_ACTION

ACTION Act01_Status:
Axis.ReadStatus();

;

IF Axis.Status.Error  THEN
	Error := TRUE;
	ErrorMessage := 'Axis Error';
	ErrorID := Axis.Status.ErrorID;
ELSIF Axis.NcToPlc.ActPos > MaxPressPosition THEN
	Error := TRUE;
	ErrorMessage := 'Axis Position lager then max position';
	ErrorID := 10;
ELSIF Option.Velocity <=0 THEN
	Error := TRUE;
	ErrorMessage := 'Axis absoulte motion Velo set error in option params';
	ErrorID := 11;
ELSIF Option.FastReachVelo <=0 THEN
	Error := TRUE;
	ErrorMessage := 'Axis fast Reach motion Velo set error in option params';
	ErrorID := 12;
ELSIF Option.BufferVelo <=0 THEN
	Error := TRUE;
	ErrorMessage := 'Axis buffer motion Velo set error in option params';
	ErrorID := 13;
ELSIF Actual_Torque  > (DeadZone_Max + 300) AND (eWorkStep =100 OR eWorkStep = 200) THEN
	Error := TRUE;
	ErrorMessage := 'Axis StartPressPosition lager then max Torque';
	ErrorID := 14;
END_IF

CASE eErrorStep OF
0:
	IF Error THEN	
		eErrorStep := 100;
	END_IF
	
100:
	mcStop.Execute := TRUE;
	IF Axis.Status.NotMoving THEN
		mcStop.Execute := FALSE;
		eErrorStep := 200;
	END_IF
	
200:
	mcStop.Execute := FALSE;
	IF NOT Error THEN;
		eErrorStep := 0;
	END_IF
END_CASE
END_ACTION

ACTION Act02_ToqueMove:
(*IF EnablePID=TRUE THEN
	ErrorTorque:=Target_Torque-Actual_Torque;;
	IF Actual_Torque< Target_Torque*0.01 THEN	(*快速下降区*)
		fPIDVelocity:=Option.FastReachVelo;
	ELSIF Actual_Torque>=Target_Torque*0.02 AND ErrorTorque>Target_Torque*0.02 THEN	(*缓冲区*)
		fPIDVelocity:=Option.BufferVelo;						(*系数需要调节*)
	ELSIF ErrorTorque>DeadZone THEN				(*精确调整区*)
		fPIDVelocity:=ErrorTorque*0.00001;		(*系数需要调节*)
	ELSIF ABS(ErrorTorque)<=DeadZone THEN		(*死区*)
		fPIDVelocity:=0;
	ELSIF ErrorTorque<-DeadZone THEN			(*过冲回调区*)
		fPIDVelocity:=ErrorTorque*0.002;		(*系数需要调节*)
	END_IF
ELSE
	fPIDVelocity:=0;
END_IF
*)

IF EnablePID=TRUE THEN
	ErrorTorque:=Target_Torque-Actual_Torque;;
	IF Actual_Torque< Target_Torque*0.005 THEN	(*快速下降区*)
		fPIDVelocity:=Option.FastReachVelo;
	ELSIF Actual_Torque>=Target_Torque*0.03*Press_Fast_xs AND ErrorTorque>Press_Slow_xs*Target_Torque*0.03 THEN	(*缓冲区*)
		fPIDVelocity:=Option.BufferVelo;						(*系数需要调节*)
	ELSIF ErrorTorque>DeadZone THEN				(*精确调整区*)
		fPIDVelocity:=ErrorTorque*0.0001;		(*系数需要调节*)
	ELSIF ABS(ErrorTorque)<=DeadZone THEN		(*死区*)
		fPIDVelocity:=0;
	ELSIF ErrorTorque<-DeadZone THEN			(*过冲回调区*)
		fPIDVelocity:=ErrorTorque*0.0005;		(*系数需要调节*)
	END_IF
ELSE
	fPIDVelocity:=0;
END_IF


CASE eTorqueStep OF
0:
	IF EnablePID THEN
		eTorqueStep := 1000;
	END_IF
	
(*实际压力与设定压力比较*)	
1000:
	mcStop.Execute := FALSE;
	IF 		fPIDVelocity > 0 THEN MoveVel.Execute := FALSE; eTorqueStep := 1200;
	ELSIF 	fPIDVelocity = 0 THEN MoveVel.Execute := FALSE; eTorqueStep := 1300;
	ELSIF 	fPIDVelocity < 0 THEN MoveVel.Execute := FALSE; eTorqueStep := 1400;
	END_IF

(*下压*)	
1200:
	MoveVel.Direction:=MC_Positive_Direction;
	MoveVel.BufferMode:=MC_BlendingNext;
	MoveVel.Velocity :=ABS(fPIDVelocity) ;
	MoveVel.Execute := TRUE;
	eTorqueStep := 1000;
	
(*停止*)	
1300:
	mcStop.Execute := TRUE;
	IF Axis.Status.NotMoving THEN
		mcStop.Execute := FALSE;
		eTorqueStep := 1000;
	END_IF 
	
(*上抬*)	
1400:
	MoveVel.Direction:=MC_Negative_Direction;
	MoveVel.BufferMode:=MC_BlendingNext;
	MoveVel.Velocity :=ABS(fPIDVelocity) ;
	MoveVel.Execute := TRUE;
	eTorqueStep := 1000;	
END_CASE
END_ACTION

ACTION Act10_Auto:
error_ton(PT:=T#30S);
Stop_ton(PT:=T#100MS);
Axis1_TON(PT:=T#20S);

	IF eWorkStep = 1250  THEN
	IF NOT Axis1_TON.Q THEN
		Axis1_TON.IN:=TRUE;
	ELSE
		Error:=TRUE;
	END_IF
ELSE
	    Axis1_TON.IN:=FALSE;
END_IF



//触发条件
rtStart(CLK:=Start_Torque , Q=> );
CASE eWorkStep OF
0:
	CurrentPressTime := T#0MS;
	Pressing := FALSE;	
	Busy := FALSE;
	MoveAbs.Execute := FALSE;
	Stop_ton.IN:=FALSE;
	tOutTime(IN:=FALSE);
	IF 	rtStart.Q THEN
		Busy := TRUE;
		Done:= FALSE;
	    HoldOK := FALSE;
		mcStop.Execute := FALSE;
		Start_Torque:=FALSE;
		eWorkStep := 20;
	END_IF

20://下压安全条件
	IF Press_condition AND NOT Error1 AND Axis.Status.ControlLoopClosed  THEN
		eWorkStep := 100;
		ELSE
		eWorkStep := 0;
		Error1:=TRUE;
	END_IF


	
(*运动到预压初始位置*)	
100:
	MoveAbs.Position := StartPressPosition ;
	MoveAbs.Velocity := Option.Velocity;
	MoveAbs.Acceleration := Option.Acc;
	MoveAbs.Deceleration := Option.Dec;
	MoveAbs.Jerk := Option.Jerk;
	MoveAbs(Execute:= TRUE ,Axis:= Axis);
	IF 	Axis.Status.NotMoving AND ABS(Axis.NcToPlc.ActPos-StartPressPosition)<0.01 THEN
		MoveAbs(Execute:= FALSE ,Axis:= Axis);
		eWorkStep := 200;
	END_IF

(*判读是否达到设定压力的范围*)	
200:	
	EnablePID := TRUE;
	error_ton.IN:=EnablePID;
	tOutTime(IN:= TRUE, PT:=T#40S , Q=> , ET=> );
	IF Actual_Torque >= DeadZone_Min AND Actual_Torque <= DeadZone_Max THEN
		eWorkStep := 1000;
		error_ton.IN:=FALSE;
	ELSIF tOutTime.Q OR Axis.Status.SoftLimitMaxExceeded THEN
		Pressing := FALSE;
		eTorqueStep := 0;
		EnablePID := FALSE;
		MoveVel.Execute := FALSE;
		mcStop.Execute := FALSE;
		HoldOK := TRUE;
		Error := TRUE;
		tonHoldPress.IN := FALSE;
		tOutTime(IN:=FALSE);
		eWorkStep := 1200;
	END_IF
	
(*保压中*)
1000:
	error_ton.IN:=FALSE;
	Pressing := TRUE;
 	tonHoldPress.IN := TRUE;
	CurrentPressTime := tonHoldPress.ET;
	IF tonHoldPress.Q THEN
		CurrentPressTime:= tonHoldPress.PT;
		Pressing := FALSE;
		eTorqueStep := 0;
		EnablePID := FALSE;
		MoveVel.Execute := FALSE;
		mcStop.Execute := FALSE;
		tonHoldPress.IN := FALSE;
		HoldOK := TRUE;
		eWorkStep := 1200;
	ELSIF Axis.Status.SoftLimitMaxExceeded THEN
		Pressing := FALSE;
		eTorqueStep := 0;
		EnablePID := FALSE;
		MoveVel.Execute := FALSE;
		mcStop.Execute := FALSE;
		HoldOK := TRUE;
		Error := TRUE;
		tonHoldPress.IN := FALSE;
		eWorkStep := 1200;
	END_IF

1100:
	MoveAbs.Execute:=FALSE;
	mcStop.Execute := TRUE;
	IF mcStop.Done THEN
		mcStop.Execute := FALSE;
		eWorkStep := 1150;
	END_IF
	
1150:
	IF //AxisArr[1].Status.NotMoving 
        Axis.Status.NotMoving   THEN
		mcStop.Execute := FALSE;
		eWorkStep := 1200;
	END_IF
	
(*升降电机返回初始位置*)	

1200:
	mcStop.Execute := TRUE;
	EnablePID:=FALSE;
	eTorqueStep := 0;
	Stop_ton.IN:=TRUE;
	IF Stop_ton.Q THEN
		eWorkStep := 1250;
	END_IF

1250:
	mcStop.Execute := FALSE;
	MoveAbs.Position := InitPosition ;
	MoveAbs.Velocity := Option.Velocity; 
	MoveAbs.Acceleration := Option.Acc;
	MoveAbs.Deceleration := Option.Dec;
	MoveAbs.Jerk := Option.Jerk;
	MoveAbs.BufferMode := MC_Aborting;
	MoveAbs.Execute := TRUE;
	BlowPermit:=TRUE;//吹气允许
	Stop_ton.IN:=FALSE;
	IF 	Axis.Status.NotMoving AND ABS(Axis.NcToPlc.ActPos-InitPosition)<0.01 THEN
		BlowPermit:=FALSE;//吹气允许
		MoveAbs.Execute := FALSE;
		eWorkStep := 1300;
	END_IF
	
1300:
	Done:= TRUE;
	Busy := FALSE;
	IF NOT Start_Torque THEN
		eWorkStep := 0;
	END_IF	 
END_CASE
END_ACTION

END_FUNCTION_BLOCK

// ---- P3POUs/P3FB/FB_DataXMLP3_Old.TcPOU
FUNCTION_BLOCK FB_DataXMLP3_Old
VAR_INPUT
    	bSave:BOOL;
	    bRead:BOOL;

END_VAR
VAR_OUTPUT
    	bSaveParDone      :BOOL;
	    bReadParDone     :BOOL;
		bError                     :BOOL;		
END_VAR

VAR


	iDataSetp: INT;
	TON10:Tc2_Standard.TON;
	I1: INT;
	rt100:Tc2_Standard.R_TRIG;
	rt101:Tc2_Standard.R_TRIG;
	bExecute1: BOOL;
	bExecute2: BOOL;


	bSaveTemp: BOOL;
	bReadTemp: BOOL;

 fbXmlSrvWrite         : FB_XmlSrvWrite;
// fbXmlSrvWrite         : FB_SrvWrite;
   bExecuteW1             : BOOL;
   sFilePathPar_W       : T_MaxString ;

 
fbXmlSrvRead   : FB_XmlSrvRead;
//fbXmlSrvRead   : FB_SrvRead;
   bExecuteR          : BOOL;
   sFilePathPar_R      : T_MaxString ;
   sXPathR             : T_MaxString;
	AA: INT;
	BB: INT;












	handleTemp: UDINT;
END_VAR


M_WriteOrRead();

ACTION M_WriteOrRead:
bError := fbXmlSrvWrite.bError OR   fbXmlSrvRead.bError;

rt100(CLK:=bSave , Q=> );//保存参数
rt101(CLK:=bRead , Q=> );//读取参数

IF rt100.Q THEN  //保存参数
	iDataSetp:=100;
	TON10.IN:=FALSE;
	I1:=1;
	bExecute1:=FALSE;
	bExecute2:=FALSE;
	bSave:=FALSE;
	bRead:=FALSE;
    bSaveTemp:=TRUE;
	bReadTemp:=FALSE;
	bSaveParDone:=FALSE;
END_IF

IF rt101.Q THEN  //读取参数
	iDataSetp:=100;
	TON10.IN:=FALSE;
	I1:=1;
	bExecute1:=FALSE;
	bExecute2:=FALSE;	
	bSave:=FALSE;
	bRead:=FALSE;
    bReadTemp:=TRUE;
    bSaveTemp:=FALSE;
    bReadParDone:=FALSE;
END_IF

TON10(IN:= , PT:=T#200MS , Q=> , ET=> );

CASE  iDataSetp OF 
	
 100:
				CASE I1 OF 
				  1://轴参数
					sFilePathPar_W  := 'C:\P3XML\P3arrAxisParV2.xml';
					fbXmlSrvWrite.pSymAddr:=ADR(arrAxisParV2);
					fbXmlSrvWrite.cbSymSize:=SIZEOF(arrAxisParV2);   

					sFilePathPar_R  :=  'C:\P3XML\P3arrAxisParV2.xml';
					fbXmlSrvRead.pSymAddr:=ADR(arrAxisParV2);
					fbXmlSrvRead.cbSymSize:=SIZEOF(arrAxisParV2);   
     
				  2://arrTempPar
		  		    sFilePathPar_W  := 'C:\P3XML\P3arrTempPar.xml';
					fbXmlSrvWrite.pSymAddr:=ADR(arrTempPar);
					fbXmlSrvWrite.cbSymSize:=SIZEOF(arrTempPar);     

					sFilePathPar_R  := 'C:\P3XML\P3arrTempPar.xml';
					fbXmlSrvRead.pSymAddr:=ADR(arrTempPar);
					fbXmlSrvRead.cbSymSize:=SIZEOF(arrTempPar);   

				  3://P3par
		  		     sFilePathPar_W  := 'C:\P3XML\P3par.xml';
					fbXmlSrvWrite.pSymAddr:=ADR(P3par);
					fbXmlSrvWrite.cbSymSize:=SIZEOF(P3par);     

					sFilePathPar_R  := 'C:\P3XML\P3par.xml';
					fbXmlSrvRead.pSymAddr:=ADR(P3par);
					fbXmlSrvRead.cbSymSize:=SIZEOF(P3par);   
					
			     4://P3par
		  		     sFilePathPar_W  := 'C:\P3XML\P3User2_Par.xml';
					fbXmlSrvWrite.pSymAddr:=ADR(P3User2_Par);
					fbXmlSrvWrite.cbSymSize:=SIZEOF(P3User2_Par);     

					sFilePathPar_R  := 'C:\P3XML\P3User2_Par.xml';
					fbXmlSrvRead.pSymAddr:=ADR(P3User2_Par);
					fbXmlSrvRead.cbSymSize:=SIZEOF(P3User2_Par);   				
			
				END_CASE
        IF  bSaveTemp THEN
              handleTemp:=fbXmlSrvWrite.handle;
   	          iDataSetp:=200;
       END_IF
        IF  bReadTemp THEN
              handleTemp:=fbXmlSrvRead.handle;
   	          iDataSetp:=300;
       END_IF

	   
	200:	//保存数据
		bExecute1:=TRUE;
        iDataSetp:=210;
	210:	
       IF  NOT fbXmlSrvWrite.bError  AND NOT fbXmlSrvWrite.bBusy AND handleTemp<>fbXmlSrvWrite.handle  THEN
             iDataSetp:=500;
      END_IF
	  
	300:	//读取参数
		bExecute2:=TRUE;
        iDataSetp:=310;
	310:	
       IF  NOT fbXmlSrvRead.bError  AND NOT fbXmlSrvRead.bBusy AND handleTemp<>fbXmlSrvRead.handle  THEN
             iDataSetp:=500;
      END_IF


	500://继续写下个文件
	  IF I1>=1 AND I1<4 THEN
		 I1:=I1+1; 
		 iDataSetp:=100; 
		 bExecute1:=FALSE; 
		 bExecute2:=FALSE; 
	  ELSIF I1>=4 THEN
          IF  bSaveTemp THEN
               bSaveParDone:=TRUE;
         END_IF

          IF  bReadTemp THEN
               bReadParDone:=TRUE;
         END_IF

		  bReadTemp:=FALSE;
          bSaveTemp:=FALSE;

	   	 iDataSetp:=666;   
	  END_IF
END_CASE


AA:=BB;

fbXmlSrvWrite(
   nMode           := XMLSRV_ADDMISSING,
   pSymAddr        :=,//ADR(Value1)
   cbSymSize       := ,//SIZEOF(Value1)
   sFilePath       := sFilePathPar_W,
   sXPath	       := '/dataentry/value',
   bExecute        := bExecute1
);


fbXmlSrvRead(
   pSymAddr       := ,
   cbSymSize      := ,
   sFilePath      := sFilePathPar_R,
   sXPath	         := '/dataentry/value',
   bExecute       := bExecute2
);
END_ACTION

END_FUNCTION_BLOCK

// ---- P3POUs/P3FB/FB_Press.TcPOU
FUNCTION_BLOCK FB_Press
VAR_IN_OUT

AxisPressing :AXIS_REF;//扭矩轴
Press_SystemRUN  :ST_SystemRUN;//热、冷压系统
Clear_press    :BOOL;//压力清零信号
Permit_Press   :BOOL;//允许热、冷压信号
Press_Finish   :BOOL;//热、冷压完成信号

END_VAR
	
VAR_INPUT
	Step: UINT;
	AxisPress	 :INT;//扭矩轴名称
	AxisTensed	 :INT;//麦拉膜轴名称
	CylinderPress	:INT;//麦拉膜气缸名称
	Press_M          :INT;//电芯记忆名称
	Press_SV :REAL;//当前压力值
	Press_P  :REAL;//压力调节值P值
	Press_I  :REAL;//压力调节值I值
	Press_D  :REAL;//压力调节值D值
	AD_Press :INT;//压力模拟量
	Press_Factor :REAL;//扭矩系数
	Torque_Offset :REAL;//扭矩偏移量
	TorqueRamp    :REAL;//扭矩变化率 
	VelocityLimit :REAL;//扭矩速度限制
	Press_Time :INT;//保持压力时间

END_VAR

VAR_OUTPUT
	Press_PV :REAL;//当前压力值
	Torque_Act :REAL;//扭矩当前值
END_VAR

VAR
Press_H_Limit :REAL;//压力上限值
Press_L_Limit :REAL;//压力下限值
Press_max     :REAL;//压力最大值
Press_min     :REAL;//压力最小值
Press_PID_Out :REAL;//PID输出值	
FB_MC_TorqueControl_1: MC_TorqueControl;
FB_MC_MoveVelocity_1: MC_MoveVelocity;
Hot_Torque: INT;
FB_Unwinding_PID_1: Unwinding_PID;
Press_Time_Z:TIME;
Press_TON :TON;
FB_MC_Stop_1: MC_Stop;
END_VAR

Press_PV:=INT_TO_REAL(AD_Press)*4;
Press_max:=Press_SV+1000;
Press_min:=Press_SV-400;
Torque_Act:=Press_PV*Press_Factor+Torque_Offset;
FB_MC_TorqueControl_1.Torque:=REAL_TO_LREAL(Press_SV*Press_Factor);
FB_MC_TorqueControl_1.TorqueRamp:=REAL_TO_LREAL(TorqueRamp);
FB_MC_TorqueControl_1.VelocityLimitHigh:=REAL_TO_LREAL(VelocityLimit+5);
FB_MC_TorqueControl_1.VelocityLimitLow:=REAL_TO_LREAL(VelocityLimit);

FB_MC_MoveVelocity_1.Velocity:=-Press_PID_Out*REAL#0.5;
FB_MC_MoveVelocity_1.Acceleration:=FB_MC_MoveVelocity_1.Velocity*10;
FB_MC_MoveVelocity_1.Deceleration:=FB_MC_MoveVelocity_1.Velocity*10;
FB_MC_MoveVelocity_1.Jerk:=FB_MC_MoveVelocity_1.Velocity*100;
FB_MC_MoveVelocity_1.Velocity:=LIMIT(-LREAL#2,FB_MC_MoveVelocity_1.Velocity,LREAL#2);
Press_Time_Z:=INT_TO_TIME(Press_Time);

IF Press_SystemRUN.iMode=1 THEN
CASE Step OF
1://驱动电机回初始位	
IF  NOT arrAxisCtrl[AxisPress].Cmd.arrbRealPoint[1] AND NOT arrAxisCtrl[AxisPress].Status.Error AND arrAxisCtrl[AxisPress].Status.Homed 
	AND arrAxisCtrl[AxisPress].Status.Enabled AND arrAxisCtrl[AxisPress].Status.NoMoving THEN
	arrAxisCtrl[AxisPress].Cmd.iGoSetPos:=1;
END_IF 

IF arrAxisCtrl[AxisPress].Cmd.arrbRealPoint[1]	AND arrAxisCtrl[AxisPress].Status.NoMoving THEN
	Step:=5;
	Clear_press:=TRUE;//压力清零信号
END_IF

5://判断是否能热、冷压

IF Permit_Press AND NOT CellMemory[Press_M].ScanCode=2 THEN
	Step:=10;
	Clear_press:=FALSE;
END_IF


10://麦拉膜轴去张开位和麦拉膜气缸张紧
arrCyCtrl[CylinderPress].Cmd.bON:=TRUE;
IF  arrAxisCtrl[AxisPress].Cmd.arrbRealPoint[1]	AND
	NOT arrAxisCtrl[AxisTensed].Cmd.arrbRealPoint[2] AND NOT arrAxisCtrl[AxisTensed].Status.Error AND arrAxisCtrl[AxisTensed].Status.Homed 
	AND arrAxisCtrl[AxisTensed].Status.Enabled AND arrAxisCtrl[AxisTensed].Status.NoMoving THEN
	arrAxisCtrl[AxisTensed].Cmd.iGoSetPos:=2;	
END_IF
 IF arrAxisCtrl[AxisTensed].Cmd.arrbRealPoint[2] AND arrAxisCtrl[AxisTensed].Status.NoMoving AND arrCyCtrl[CylinderPress].Status.ONState 
	AND NOT arrCyCtrl[CylinderPress].Status.Error1 THEN
	step:=20;
END_IF

20://扭矩轴去电芯位

IF NOT arrAxisCtrl[AxisPress].Cmd.arrbRealPoint[2] AND NOT arrAxisCtrl[AxisPress].Status.Error AND arrAxisCtrl[AxisPress].Status.Homed 
	AND arrAxisCtrl[AxisPress].Status.Enabled AND arrAxisCtrl[AxisPress].Status.NoMoving THEN
	arrAxisCtrl[AxisPress].Cmd.iGoSetPos:=2;	
END_IF 

IF arrAxisCtrl[AxisPress].Cmd.arrbRealPoint[2]	AND Permit_Press AND arrAxisCtrl[AxisPress].Status.NoMoving THEN
	Step:=30;
END_IF

30://开始走扭矩
FB_MC_TorqueControl_1.Execute:=TRUE;
IF FB_MC_TorqueControl_1.InTorque AND Press_PV>Press_min AND Press_PV<Press_max THEN//扭矩达到范围值开始走PID
	Step:=40;
	FB_MC_TorqueControl_1.Execute:=FALSE;
END_IF

40://保压
FB_MC_MoveVelocity_1.Execute:=TRUE;//走PID
Press_TON.PT:=Press_Time_Z;
Press_TON.IN:=TRUE;
IF Press_TON.Q THEN//保压时间达到后
	Step:=50;
	Press_TON.IN:=FALSE;
	FB_MC_MoveVelocity_1.Execute:=FALSE;
END_IF
	
50://轴停止
FB_MC_Stop_1.Execute:=TRUE;
IF FB_MC_Stop_1.Done THEN
	Step:=60;
	FB_MC_Stop_1.Execute:=FALSE;
END_IF

60://扭矩轴回初始位
IF  NOT arrAxisCtrl[AxisPress].Cmd.arrbRealPoint[1] AND NOT arrAxisCtrl[AxisPress].Status.Error AND arrAxisCtrl[AxisPress].Status.Homed 
	AND arrAxisCtrl[AxisPress].Status.Enabled AND arrAxisCtrl[AxisPress].Status.NoMoving THEN
	arrAxisCtrl[AxisPress].Cmd.iGoSetPos:=1;	
END_IF 
IF arrAxisCtrl[AxisPress].Cmd.arrbRealPoint[1] AND arrAxisCtrl[AxisPress].Status.NoMoving THEN
	Permit_Press :=FALSE;//复位允许冷、热压信号
	Press_Finish:=TRUE;//冷热压完成信号可以下料
	Step:=70;
END_IF

70:
Step:=1;

END_CASE
END_IF

ACTION TorqueAndPID:
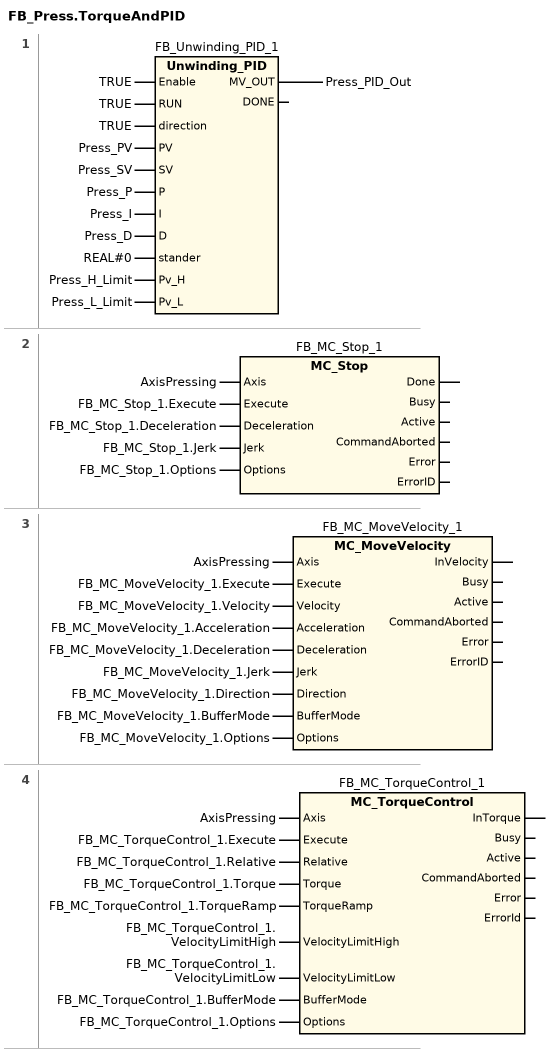
// NETWORK 1
FB_Unwinding_PID_1(
    Enable := TRUE,
    RUN := TRUE,
    direction := TRUE,
    PV := Press_PV,
    SV := Press_SV,
    P := Press_P,
    I := Press_I,
    D := Press_D,
    stander := REAL#0,
    Pv_H := Press_H_Limit,
    Pv_L := Press_L_Limit); // Unwinding_PID
Press_PID_Out := FB_Unwinding_PID_1.MV_OUT;

// NETWORK 2
FB_MC_Stop_1(
    Axis := AxisPressing,
    Execute := FB_MC_Stop_1.Execute,
    Deceleration := FB_MC_Stop_1.Deceleration,
    Jerk := FB_MC_Stop_1.Jerk,
    Options := FB_MC_Stop_1.Options); // MC_Stop

// NETWORK 3
FB_MC_MoveVelocity_1(
    Axis := AxisPressing,
    Execute := FB_MC_MoveVelocity_1.Execute,
    Velocity := FB_MC_MoveVelocity_1.Velocity,
    Acceleration := FB_MC_MoveVelocity_1.Acceleration,
    Deceleration := FB_MC_MoveVelocity_1.Deceleration,
    Jerk := FB_MC_MoveVelocity_1.Jerk,
    Direction := FB_MC_MoveVelocity_1.Direction,
    BufferMode := FB_MC_MoveVelocity_1.BufferMode,
    Options := FB_MC_MoveVelocity_1.Options); // MC_MoveVelocity

// NETWORK 4
FB_MC_TorqueControl_1(
    Axis := AxisPressing,
    Execute := FB_MC_TorqueControl_1.Execute,
    Relative := FB_MC_TorqueControl_1.Relative,
    Torque := FB_MC_TorqueControl_1.Torque,
    TorqueRamp := FB_MC_TorqueControl_1.TorqueRamp,
    VelocityLimitHigh := FB_MC_TorqueControl_1.VelocityLimitHigh,
    VelocityLimitLow := FB_MC_TorqueControl_1.VelocityLimitLow,
    BufferMode := FB_MC_TorqueControl_1.BufferMode,
    Options := FB_MC_TorqueControl_1.Options); // MC_TorqueControl
END_ACTION

END_FUNCTION_BLOCK

// ---- P3POUs/P3FB/Unwinding_PID.TcPOU
FUNCTION_BLOCK Unwinding_PID
VAR_INPUT
	Enable:BOOL;
	RUN:BOOL;//模块的使能
	direction:BOOL;//方向选择
	PV:REAL;//过程值
	SV:REAL;//设定值
	P:REAL := 0.0;//P参数
	I:REAL := 0.0;//I参数
	D:REAL := 0.0;//D参数
	stander: REAL := 30.0;//残差标准量	
	Pv_H:REAL;//过程值的最大值
	Pv_L:REAL;//过程值的最小值
END_VAR
VAR_OUTPUT
	MV_OUT:REAL;//MV输出值
	DONE:BOOL;//计算完成
END_VAR
VAR
	
	Total: REAL;
	DATA011: REAL;
	DATA01: REAL;
	DATA021: REAL;
	DATA02: REAL;
	DATA03: REAL;
	DATA031: REAL;
	Ek: REAL;
	Pvalue: REAL;
	R_TRIG_instance: R_TRIG;
	PD_Control: BOOL;
	Trigger: BOOL;
	Ivalue: REAL;
	PID_Control: BOOL;
	R_TRIG_instance1: R_TRIG;
	Trigger1: BOOL;
	D_Point: REAL;
	Dvalue: REAL;
	MV: REAL;
END_VAR

IF Enable THEN
	DONE:=TRUE;
	DATA011:=100.00*(Pv_H-SV)/(Pv_H-Pv_L);
	DATA01:=ABS(DATA011);
	DATA021:=100.00*(SV-Pv_L)/(Pv_H-Pv_L);
	DATA02:=ABS(DATA021);
	DATA03:=Min(DATA01,DATA02);
	DATA031:=300*DATA03;
  IF RUN=TRUE THEN
	Ek:=(SV-PV)*100.00/(Pv_H-Pv_L); //	转换为0-300
	Pvalue:=P*Ek;
 	R_TRIG_instance(CLK:=PD_Control , Q=> Trigger);
	IF Trigger THEN 
	 Total:=0.0;
	 Ivalue:=0.0;
    END_IF; 
	IF PID_Control=TRUE THEN
		Total:=Total+Ek;
		IF Total>=DATA031	 THEN
			Total:=DATA031;
		END_IF;
		IF Total<-(DATA031) THEN
			Total:=-(DATA031);
		END_IF;
		Ivalue:=I*Total/100.00;  //100.00;  //I值放大100倍
	END_IF;
	R_TRIG_instance1(CLK:=PD_Control , Q=> Trigger1);
	IF Trigger1=TRUE THEN
			D_Point:=0.0;
		END_IF;
	Dvalue:=D*(Ek-D_Point);
	D_Point:=Ek;
	IF (ABS(Ek)-stander)>0.0 THEN
		PD_Control:=TRUE; 
		PID_Control:=FALSE;
	ELSIF (ABS(Ek)-stander)<0.0 THEN
		PID_Control:=TRUE;
		PD_Control:=FALSE; 
	END_IF;
	IF PD_Control THEN
		MV:=100*(Pvalue+Dvalue)/(DATA03*100.00+DATA03*D);
	ELSIF PID_Control THEN
		MV:=100*(Pvalue+Dvalue)/(DATA03*100.00+DATA03*D)+100*Ivalue/(DATA031);
	END_IF;
  END_IF;
  IF direction=FALSE THEN
	  MV_OUT:=LIMIT(REAL#-100.00,MV,REAL#100.00);
  ELSE
	  MV_OUT:=-(LIMIT(REAL#-100.00,MV,REAL#100.00));
  END_IF; 	
ELSE
	Total:=0.00;
	MV_OUT:=0.00;
	DONE:=FALSE;	
END_IF

END_FUNCTION_BLOCK

// ---- P3POUs/P3FB/FB_PulsPercentage.TcPOU
FUNCTION_BLOCK FB_PulsPercentage
VAR_INPUT
	fPercentage :INT; 
    iTimeBasic :INT;//时 基  1S
 
END_VAR
VAR_OUTPUT
	bDOPuls:BOOL;

END_VAR
VAR
	ton01:Tc2_Standard.TON;
    tonON:Tc2_Standard.TON;
    tonOFF:Tc2_Standard.TON;

	iStep: INT;
	AA1: INT;
END_VAR

 
ton01(IN:= , PT:= INT_TO_TIME(iTimeBasic*1000), Q=> , ET=> ); //单位S
tonON(IN:= , PT:= , Q=> , ET=> );
tonOFF(IN:= , PT:=, Q=> , ET=> );

IF NOT ton01.Q THEN
	ton01.IN:=TRUE;
END_IF

IF  ton01.Q THEN
	ton01.IN:=FALSE;
	iStep:=10;
END_IF


//  AA1:= REAL_TO_INT (fPercentage*iTimeBasic*1000/100) ;

 
CASE iStep OF 	
	
10:  //输出ON
 tonON.PT:= INT_TO_TIME ( REAL_TO_INT (fPercentage*iTimeBasic*1000/100) );
 IF tonON.PT>=T#10MS THEN
	 bDOPuls:=TRUE; 
	 tonON.IN:=TRUE;
	 iStep:=20;
  ELSE
	 bDOPuls:=FALSE; 
	 tonON.IN:=FALSE;
	 iStep:=100;  
 END_IF
20:  //输出ON 
  IF tonON.Q THEN
	  bDOPuls:=FALSE;
	  tonON.IN:=FALSE; 
	  iStep:=100;
  END_IF

100: //输出OFF


END_CASE

END_FUNCTION_BLOCK

// ---- P3POUs/P3FB/Oven_button.TcPOU
FUNCTION_BLOCK Oven_button

VAR_IN_OUT
	Oven_Button :ARRAY[1..42] OF BOOL;
	Oven_Flow   :ARRAY[1..42] OF BOOL;
END_VAR


VAR_INPUT
END_VAR


VAR_OUTPUT
END_VAR



VAR
	step :UINT;
	a :INT;
	i:INT;
END_VAR

IF P3_SystemRUN.iMode=3 THEN
	



IF arrAxisCtrlV2[P3AxisNo.P3_M2_OvenRetracting].Status.Error OR arrAxisCtrlV2[P3AxisNo.P3_M2_OvenCarrying].Status.Error OR arrAxisCtrlV2[P3AxisNo.P3_M2_OvenUpDown].Status.Error THEN
step:=9999;
END_IF

IF step=9999 AND P3_SystemRUN.btnReset THEN
	step:=0;
END_IF

CASE step OF
0:
	IF NOT arrAxisCtrlV2[P3AxisNo.P3_M2_OvenRetracting].Status.Error AND NOT arrAxisCtrlV2[P3AxisNo.P3_M2_OvenCarrying].Status.Error AND NOT arrAxisCtrlV2[P3AxisNo.P3_M2_OvenUpDown].Status.Error
	AND Oven_button[a] THEN
		step:=10;
		Oven_button[a]:=FALSE;
	END_IF

10://P3_M2烤箱上料夹进退电机去初始位
	IF NOT arrAxisCtrlV2[P3AxisNo.P3_M2_OvenRetracting].Cmd.arrbRealPoint[43] AND NOT arrAxisCtrlV2[P3AxisNo.P3_M2_OvenRetracting].Status.Error AND arrAxisCtrlV2[P3AxisNo.P3_M2_OvenRetracting].Status.Homed 
		AND arrAxisCtrlV2[P3AxisNo.P3_M2_OvenRetracting].Status.Enabled AND arrAxisCtrlV2[P3AxisNo.P3_M2_OvenRetracting].Status.NoMoving THEN
		arrAxisCtrlV2[P3AxisNo.P3_M2_OvenRetracting].Cmd.iGoSetPos:=43;
	END_IF
	IF  arrAxisCtrlV2[P3AxisNo.P3_M2_OvenRetracting].Cmd.arrbRealPoint[43]  AND Oven_POS1  AND arrAxisCtrlV2[P3AxisNo.P3_M2_OvenRetracting].Status.NoMoving THEN
		step:=20;	
	END_IF

20://P3_M2烤箱上料夹升降电机去初始位
	IF  arrAxisCtrlV2[P3AxisNo.P3_M2_OvenRetracting].Cmd.arrbRealPoint[43] AND
		NOT arrAxisCtrlV2[P3AxisNo.P3_M2_OvenUpDown].Cmd.arrbRealPoint[43] AND NOT arrAxisCtrlV2[P3AxisNo.P3_M2_OvenUpDown].Status.Error AND arrAxisCtrlV2[P3AxisNo.P3_M2_OvenUpDown].Status.Homed 
		AND arrAxisCtrlV2[P3AxisNo.P3_M2_OvenUpDown].Status.Enabled AND arrAxisCtrlV2[P3AxisNo.P3_M2_OvenUpDown].Status.NoMoving THEN
		arrAxisCtrlV2[P3AxisNo.P3_M2_OvenUpDown].Cmd.iGoSetPos:=43;	
	END_IF
	
	IF  arrAxisCtrlV2[P3AxisNo.P3_M2_OvenUpDown].Cmd.arrbRealPoint[43] AND arrAxisCtrlV2[P3AxisNo.P3_M2_OvenUpDown].Status.NoMoving THEN
		
		
	step:=30;	
	END_IF
	
30:	//P3_M2烤箱上料夹平移电机去烘烤a位
	IF  arrAxisCtrlV2[P3AxisNo.P3_M2_OvenUpDown].Cmd.arrbRealPoint[43] AND  arrAxisCtrlV2[P3AxisNo.P3_M2_OvenRetracting].Cmd.arrbRealPoint[43] AND 
		NOT arrAxisCtrlV2[P3AxisNo.P3_M2_OvenCarrying].Cmd.arrbRealPoint[a] AND NOT arrAxisCtrlV2[P3AxisNo.P3_M2_OvenCarrying].Status.Error AND arrAxisCtrlV2[P3AxisNo.P3_M2_OvenCarrying].Status.Homed 
		AND arrAxisCtrlV2[P3AxisNo.P3_M2_OvenCarrying].Status.Enabled AND arrAxisCtrlV2[P3AxisNo.P3_M2_OvenCarrying].Status.NoMoving THEN
		arrAxisCtrlV2[P3AxisNo.P3_M2_OvenCarrying].Cmd.iGoSetPos:=a;	
	END_IF
	
	IF  arrAxisCtrlV2[P3AxisNo.P3_M2_OvenCarrying].Cmd.arrbRealPoint[a] AND arrAxisCtrlV2[P3AxisNo.P3_M2_OvenCarrying].Status.NoMoving THEN
		
	step:=40;	
	END_IF


40://P3_M2烤箱上料夹升降电机去烘烤a位
	IF  arrAxisCtrlV2[P3AxisNo.P3_M2_OvenRetracting].Cmd.arrbRealPoint[43] AND
		NOT arrAxisCtrlV2[P3AxisNo.P3_M2_OvenUpDown].Cmd.arrbRealPoint[a] AND NOT arrAxisCtrlV2[P3AxisNo.P3_M2_OvenUpDown].Status.Error AND arrAxisCtrlV2[P3AxisNo.P3_M2_OvenUpDown].Status.Homed 
		AND arrAxisCtrlV2[P3AxisNo.P3_M2_OvenUpDown].Status.Enabled AND arrAxisCtrlV2[P3AxisNo.P3_M2_OvenUpDown].Status.NoMoving THEN
		arrAxisCtrlV2[P3AxisNo.P3_M2_OvenUpDown].Cmd.iGoSetPos:=a;	
	END_IF
	
	IF  arrAxisCtrlV2[P3AxisNo.P3_M2_OvenUpDown].Cmd.arrbRealPoint[a] AND arrAxisCtrlV2[P3AxisNo.P3_M2_OvenUpDown].Status.NoMoving THEN
		Oven_Flow[a]:=TRUE;
	step:=50;	
	END_IF
END_CASE
END_IF

END_FUNCTION_BLOCK

// ---- P3POUs/P3FB/Oven_Time.TcPOU
FUNCTION_BLOCK Oven_Time
VAR_IN_OUT
	Oven_Cell :ARRAY[1..42] OF BOOL;//烤箱电芯记忆
	Oven_Finish :ARRAY[1..42] OF BOOL;//烤箱完成信号
	Oven_shijian :TIME;//设定时间
	T_achieve :ARRAY[1..42] OF BOOL;//温度达到信号
	Ovencell_Shield :ARRAY[1..42] OF BOOL;//烤箱电芯屏蔽
	Oven_JS :ARRAY[1..42] OF UDINT;//加热完成计数（每10S计数一次）
	
END_VAR
VAR_INPUT
END_VAR
VAR_OUTPUT
Residue_T :ARRAY[1..42] OF UDINT;	
END_VAR
VAR
Oven_time :ARRAY[1..42] OF Tc2_Standard.TON;
Oven_shijian_Z :ARRAY[1..42] OF TIME;
K :INT:=1;
T_Residue :ARRAY[1..42] OF TIME;
JS_ton :ARRAY[1..42] OF Tc2_Standard.TON;
END_VAR


K:=K+1;
IF K<1 OR K>42 THEN
	K:=1;
END_IF
T_Residue[K]:=Oven_time[K].ET;
Residue_T[K]:=TIME_TO_UDINT(T_Residue[K]/60000);
Oven_shijian_Z[K] :=Oven_shijian;
Oven_time[K](IN:=(Oven_Cell[K] AND NOT Ovencell_Shield[K] (*AND T_achieve[K]*)),PT:=Oven_shijian_Z[K]);
IF Oven_Cell[K] (*AND T_achieve[K]*) AND Oven_time[K].Q AND NOT Ovencell_Shield[K] THEN
	Oven_Finish[K]:=TRUE;

END_IF


JS_ton[K](PT:=T#5S);
IF Oven_Finish[K] AND Oven_Cell[K] AND NOT Ovencell_Shield[K] THEN
	IF JS_ton[K].Q THEN
		JS_ton[K].IN:=FALSE;
		Oven_JS[K]:=Oven_JS[K]+1;
	ELSE
		JS_ton[K].IN:=TRUE;
	END_IF
END_IF


IF Oven_Finish[K] AND Oven_Cell[K] AND  Ovencell_Shield[K] THEN
	JS_ton[K].IN:=FALSE;
	Oven_JS[K]:=0;
END_IF

IF NOT Oven_Cell[K] THEN
	JS_ton[K].IN:=FALSE;
	Oven_JS[K]:=0;
	Oven_Finish[K]:=FALSE;
END_IF

END_FUNCTION_BLOCK

// ---- P3POUs/P3FB/FB_SetMoter_auto.TcPOU
FUNCTION_BLOCK FB_SetMoter_auto
VAR_INPUT
Home_done		:BOOL;//排杆电机回零完成	
biSensor        :BOOL;//对射感应
P_OT			:BOOL;//上限感应
N_OT			:BOOL;//下限感应
bHave			:BOOL;//有料感应
Box				:BOOL;//有料盒感应
END_VAR
VAR_OUTPUT
Full			:BOOL;//满料信号	
END_VAR
VAR_IN_OUT
bHome      	 	:BOOL;//回零信号

Push_NG     	:BOOL;//放NG料中
bGoWorkPos		:BOOL;//上升定位
bLeaveWorkPos	:BOOL;//下降定位

JOG_N			:BOOL;//下降
JOG_P			:BOOL;//上升	
END_VAR
VAR
UP_ton :Tc2_Standard.TON;
Down_ton :Tc2_Standard.TON;
Step_NG         :UINT;
Step_1			:UINT;
	home_ton: Ton;
END_VAR

IF biSensor AND N_OT THEN
	//Step_NG:=666;
	Full:=TRUE;
ELSIF Full AND NOT bHave THEN
	Full:=FALSE;	
END_IF

UP_ton(PT:=T#2S);
Down_ton(PT:=T#2S);
home_ton(PT:=T#500MS);


	
CASE Step_NG OF

0:
IF 	Home_done AND biSensor  AND NOT Full  AND Box AND Step_1=0 AND NOT Push_NG THEN
	Step_NG:=10;
END_IF


10:
	JOG_N:=TRUE;
	JOG_P:=FALSE;
	IF NOT biSensor THEN
		JOG_N:=FALSE;
		JOG_P:=FALSE;
		Step_NG:=20;
	END_IF

20:
	JOG_P:=FALSE;
	JOG_N:=FALSE;
	Step_NG:=0;

END_CASE


CASE Step_1 OF
0:
	IF 	NOT Home_done THEN
		Step_1:=10;
		Step_NG:=0;
		home_ton.IN:=FALSE;
	END_IF

10:
	IF Home_done AND biSensor THEN
		Step_1:=20;
		
	END_IF

20:
	home_ton.IN:=TRUE;
	IF home_ton.Q THEN
		Step_1:=0;
		home_ton.IN:=FALSE;
	END_IF

END_CASE

END_FUNCTION_BLOCK

// ---- P3POUs/P3FB/Sampling.TcPOU
FUNCTION_BLOCK Sampling



VAR_INPUT
	S_start  :BOOL;//采集触发条件
	S_amount :UINT:=3;//采集次数
	S_site   :REAL ;//采集地址
	S_time   :REAL;//采集时间间隔
END_VAR

VAR_IN_OUT
	S_finish :BOOL;//采集完成	
END_VAR

VAR_OUTPUT
	Result_mean :REAL;//平均值
END_VAR




VAR
	a :UINT:=1;
	Sam_sum :REAL;//采样总值
	Sam_max :REAL;//采样最大值
	Sam_min :REAL;//采样最小值
	Cache_data :ARRAY[1..36000] OF  REAL;
	Sam_step :UINT;
	Sam_ton :Tc2_Standard.TON;
	S_time1 :TIME;
	Out_max :REAL;
END_VAR

S_time1:=REAL_TO_TIME(S_time*1000);
Sam_ton(PT:=S_time1);

IF S_amount>36000 THEN
	S_amount:=36000;
END_IF



CASE Sam_step OF
0:
IF 	S_start AND NOT S_finish THEN
	Result_mean:=0;
	a:=1;
	Sam_sum:=0;
	MEMSET(ADR(Cache_data),0,SIZEOF(Cache_data));
	Sam_step:=10;
END_IF

10:
IF a=(S_amount+1) THEN
	Sam_step:=500;
	ELSIF a<(S_amount+1) THEN
	Sam_step:=100;
END_IF

100:
Cache_data[a]:=S_site;
Sam_ton.IN:=TRUE;
Sam_step:=105;

105:
IF a=1 THEN
Sam_max:=Cache_data[a];	
Sam_min:=Cache_data[a];
Sam_step:=110;	
ELSE
Sam_step:=110;
END_IF


110:
IF Sam_ton.Q THEN
	Sam_step:=120;
	Sam_ton.IN:=FALSE;
END_IF

120:
IF Sam_max<Cache_data[a] THEN
	Sam_max:=Cache_data[a];
	Sam_step:=130;
	ELSE
	Sam_step:=130;
END_IF

130:

IF Sam_min>Cache_data[a] THEN
	Sam_min:=Cache_data[a];
	Sam_step:=140;
	ELSE
	Sam_step:=140;
END_IF


140:
Sam_sum:=Sam_sum+Cache_data[a];
a:=a+1;
Sam_step:=150;

150:
Sam_step:=10;

500:
Sam_sum:=(Sam_sum-Sam_max-Sam_min);
Sam_step:=510;

510:
Result_mean:=Sam_sum/(a-3);
S_finish:=TRUE;
Sam_step:=0;





END_CASE

END_FUNCTION_BLOCK
